FUNCTION_BLOCK F_Scale
VAR_INPUT
	RawData					:	LREAL;
	
	RawDataLowerOffLimit	:	LREAL;
	RawDataUpperLimit		:	LREAL;
	
	ScaleDataLowerOffLimit	:	LREAL;
	ScaleDataUpperLimit		:	LREAL;
END_VAR
VAR_OUTPUT
END_VAR
VAR
END_VAR

END_FUNCTION_BLOCK

(* stored: Version 1.1.0.1, ProductVersion 3.1.4024.9
   POU F_Scale: Id {67b735c1-4990-4959-87c8-be02f5cb698e}, SpecialFunc None *)
